// TIA Portal V20 export
TYPE "LBP_typeMcp310StandardInput"
TITLE = MCP 310 image / Image du MCP 310
// Input image of MCP 310 / Image d'entrée du MCP 310
   STRUCT
      auto : Bool;
      mda : Bool;
      jog : Bool;
      singleBlock : Bool;
      spindleIncrease : Bool;
      spindle100 : Bool;
      spindleDecrease : Bool;
      cycleStop : Bool;
      teachIn : Bool;
      repos : Bool;
      refPoint : Bool;
      keySwitch3 : Bool;
      spindleLeft : Bool;
      spindleStop : Bool;
      spindleRight : Bool;
      cycleStart : Bool;
      inc1 : Bool;
      inc10 : Bool;
      inc100 : Bool;
      inc1000 : Bool;
      keySwitch0 : Bool;
      incVar : Bool;
      feedrateStop : Bool;
      feedrateStart : Bool;
      feedrateOvrA : Bool;
      feedrateOvrB : Bool;
      feedrateOvrC : Bool;
      feedrateOvrD : Bool;
      feedrateOvrE : Bool;
      keySwitch1 : Bool;
      keySwitch2 : Bool;
      reset : Bool;
      optionalKey1 : Bool;   // KT-IN1
      optionalKey2 : Bool;   // KT-IN2
      optionalKey3 : Bool;   // KT-IN3
      optionalKey4 : Bool;   // KT-IN4
      optionalKey5 : Bool;   // KT-IN5
      rapidTraverse : Bool;
      minus : Bool;
      plus : Bool;
      axisX : Bool;
      axisY : Bool;
      axisZ : Bool;
      axis4 : Bool;
      axis5 : Bool;
      axis6 : Bool;
      optionalKey6 : Bool;   // KT-IN6
      customerKey16 : Bool;   // T16
      customerKey15 : Bool;   // T15
      customerKey14 : Bool;   // T14
      customerKey13 : Bool;   // T13
      mcsWcs : Bool;
      customerKey12 : Bool;   // T12
      customerKey11 : Bool;   // T11
      customerKey10 : Bool;   // T10
      customerKey9 : Bool;   // T9
      customerKey8 : Bool;   // T8
      customerKey7 : Bool;   // T7
      customerKey6 : Bool;   // T6
      customerKey5 : Bool;   // T5
      customerKey4 : Bool;   // T4
      customerKey3 : Bool;   // T3
      customerKey2 : Bool;   // T2
      customerKey1 : Bool;   // T1
   END_STRUCT;
END_TYPE
